TYPE Cmp3LaneSwitchMainSim :
STRUCT
	
	//Component Sims
	SimMode: DINT := 0;
	GateActionMode: BOOL;
	GateProceedWithSingleAction: BOOL;
	ReallyLongFaultTime: BOOL;
	AutoPurgePostSwitch: BOOL;
	DBBypass: BOOL;
	IgnoreMachineReady: BOOL;

	//TC Sims
	TC_VersionToCall: DINT;
	ForceInfeedLane: cLaneSel;
	ForceOutfeedLane: cLaneSel;
	RoundRobinOutput: BOOL;
	InputLaneDisabled: ARRAY[1..3] Of BOOL;
	OutputLaneDisabled: ARRAY[1..3] OF BOOL;
	ForceRFID: BOOL;
	DestinationFIFO: ARRAY[0..2] OF cLaneSel;
	
END_STRUCT
END_TYPE

(* stored: Version 1.1.0.1, ProductVersion 3.1.4024.6
   DUT Cmp3LaneSwitchMainSim: Id {1e24b8fd-d965-4123-91a7-eef1e5f4604f} *)
